(* PLC project Unnamed, Unknown Unnamed 1 *)
(* stored: creationDateTime 2026-01-05T14:39:47, modificationDateTime 2026-01-05T14:39:47 *)

PROGRAM main
  VAR_INPUT
    X0 : BOOL;
    X1 : BOOL;
    X2 : BOOL;
  END_VAR
  VAR_OUTPUT
    Y0 : BOOL;
  END_VAR
  VAR
    M0 : BOOL;
  END_VAR

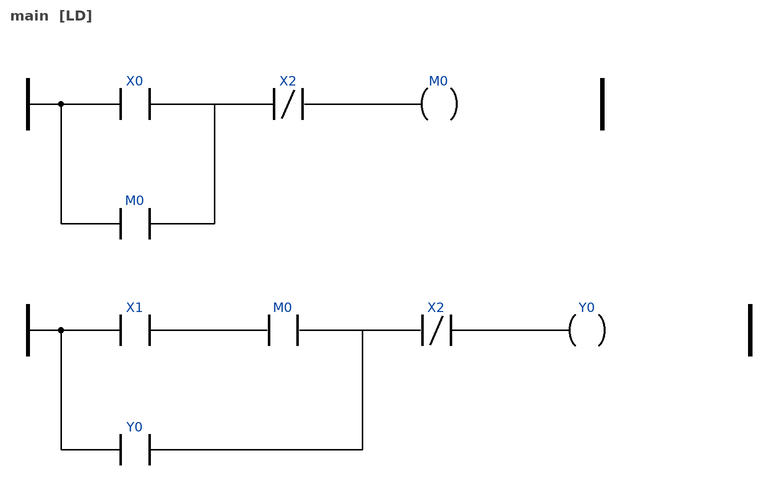
(* LD diagram, written out as Structured Text *)
M0 := (X0 OR M0) AND NOT X2;
Y0 := (X1 AND M0 OR Y0) AND NOT X2;
END_PROGRAM

CONFIGURATION Config0
  RESOURCE Res0 ON PLC
    TASK task0(INTERVAL := T#20ms, PRIORITY := 1);
    PROGRAM instance0 WITH task0 : main;
  END_RESOURCE
END_CONFIGURATION
